{attribute 'GeneratedUsingTerminal: EPP1816-3008-0016'}
{attribute addProperty BoxType "EPP1816-3008-0016"}
{attribute addProperty Id "StatusAT %I*Status_A3AA621F2ValueAT %I*INT2"}
{attribute addProperty CRC "3286137354"}
{attribute addProperty Size "4"}
TYPE AI_Inputs_Channel_C3DE7A0A :
STRUCT
	{attribute addProperty Name "Status"}
	Status AT %I* : Status_A3AA621F;
	{attribute addProperty Name "Value"}
	Value AT %I* : INT;
END_STRUCT
END_TYPE

(* stored: Version 1.2.0.0, ProductVersion 3.1.4024.9
   DUT AI_Inputs_Channel_C3DE7A0A: Id {4bacb961-96f0-4546-9743-8ea6c3fc3019} *)
